// TwinCAT 3 PLC project OCPPClient
// Title: TwinCAT IoT OCPP Client GettingStarted
// Company: Beckhoff Automation GmbH & Co. KG
// ProjectVersion: 1.0.3.0
// ProgramVersion: 3.1.4026.16
// libraries:
//   Tc2_Standard, * (Beckhoff Automation GmbH)
//   Tc2_System, * (Beckhoff Automation GmbH)
//   Tc3_OCPP, * (Beckhoff Automation GmbH)
// project tree:
//   / PlcTask.TcTTO
//   POUs/ MAIN.TcPOU
// real-time tasks:
//   TASK PlcTask: cycle T#10ms, priority 20, ADS port 350
//   TASK PlcTask1: cycle T#10ms, priority 21, ADS port 351

CONFIGURATION OCPPClient
    RESOURCE PLC ON TwinCAT3
        TASK PlcTask(INTERVAL := T#10ms, PRIORITY := 20);
        PROGRAM MAIN WITH PlcTask : MAIN;
    END_RESOURCE
END_CONFIGURATION

// ---- POUs/MAIN.TcPOU
PROGRAM MAIN
VAR
	// Client param
	stClientParam 	: ST_OCPP1_ClientParam :=(sHost:='127.0.0.1', nPort:=8080, sIdentity:='TestIdent',sPath:='ocpp',eDebugLevel:=E_OCPP_DebugLevel.MessageLogFile, eTraceLevel:=TcTraceLevel.tlVerbose); 
	fbClient 		: FB_OCPP1_Client(stClientParam, 0, 0);
	eAction 		: E_OCPP1_Action;
	hMessageId 		: T_OCPP_MessageId;
		
	// Status notification
	bSendStatus		: BOOL;
	eError			: E_OCPP1_ChargePointError;
	eStatus			: E_OCPP1_ChargePointStatus;

	// Authorize
	stIdTagInfo		: ST_OCPP1_IdTagInfo;
	sIdTag			: T_OCPP1_IdToken:='Test123';
	
	// Start transaction
	nConnectorId	: UDINT;
	nMeterStart		: UDINT;
	nTransactionId	: UDINT;
	
	//Stop transaction
	nMeterStop		: UDINT;
	
	// Charging sample
	nState			: INT;
	bStartCharging	: BOOL;
	bAuthorized		: BOOL;
	bChargingStarted: BOOL;
	bChargingStopped: BOOL;
	timerCharge		: TON:=(PT:=T#10S);
END_VAR

// Charging sample
CASE nState OF
	0: 
		IF bStartCharging THEN
			bStartCharging:=FALSE;
			eAction:=E_OCPP1_Action.Authorize;
			nState:=nState+1;
		END_IF
	1:	
		IF bAuthorized THEN
			bAuthorized:=FALSE;
			nMeterStart:=nMeterStop;
			eAction:=E_OCPP1_Action.StartTransaction;
			nState:=nState+1;
		END_IF
	2:
		IF bChargingStarted THEN
			//10 seconds charging simulation
			timerCharge(IN:=TRUE);
			IF timerCharge.Q THEN
				bChargingStarted:=FALSE;
				timerCharge(IN:=FALSE);
				nMeterStop:=nMeterStart+10;
				eAction:=E_OCPP1_Action.StopTransaction;
				nState:=nState+1;
			END_IF
		END_IF
	3: 	
		IF bChargingStopped THEN
			bChargingStopped:=FALSE;
			nState:=0;
		END_IF
END_CASE

// Send StatusNotification
IF bSendStatus THEN
	bSendStatus:=FALSE;
	eError:=E_OCPP1_ChargePointError.HighTemperature;
	eStatus:=E_OCPP1_ChargePointStatus.SuspendedEV;
	eAction:=E_OCPP1_Action.StatusNotification;
END_IF

// Different OCPP commands implemented for OCPP client
CASE eAction OF
	E_OCPP1_Action.None:
		IF NOT fbClient.bError AND fbClient.bValid THEN 
			fbClient.PollRequest(hMessageId=> hMessageId, eAction=> eAction );
		ELSE 
			// Implement error handling here		
		END_IF		
	E_OCPP1_Action.Authorize:
		IF fbClient.SendAuthorize(sIdTag:=sIdTag, eStatus => stIdTagInfo.eStatus) THEN
			IF stIdTagInfo.eStatus = E_OCPP1_AuthorizationStatus.Accepted THEN
				bAuthorized :=TRUE ;
				eAction	:= E_OCPP1_Action.None;
			END_IF
		END_IF
	E_OCPP1_Action.StartTransaction:
		IF fbClient.SendStartTransaction(sIdTag:=sIdTag, nConnectorId:=nConnectorId, nMeterStart:=nMeterStart, eStatus => stIdTagInfo.eStatus, nTransactionId => nTransactionId) THEN
			IF stIdTagInfo.eStatus = E_OCPP1_AuthorizationStatus.Accepted THEN
				bChargingStarted := TRUE;
				eAction	:= E_OCPP1_Action.None;
			END_IF
		END_IF
	E_OCPP1_Action.StopTransaction:
		IF fbClient.SendStopTransaction(nConnectorId:=nConnectorId, nMeterStop:=nMeterStop, eStatus => stIdTagInfo.eStatus) THEN
			bChargingStopped := TRUE;
			eAction	:= E_OCPP1_Action.None;
		END_IF
	E_OCPP1_Action.StatusNotification:
		IF fbClient.SendStatusNotification(nConnectorId:=nConnectorId, eError, eStatus) THEN
			eAction	:= E_OCPP1_Action.None;
		END_IF
	// Implement here more functionalities like: 
	// E_OCPP1_Action.TriggerMessage:
ELSE
	eAction := E_OCPP1_Action.None;
	// not implemented... 
END_CASE

END_PROGRAM
